REGION Network 145: PFE Maintenance Warnings_[Em5 → Em9]
   RUNG wire#powerrail
      Contact( "Unit1.Alarms".NoDataTransfer[12] )
      { S7_Templates := "time_type := Time" } "Unit1.Alarms".tonMaintenanceWarning[52].TON(pt := #DelayTime, et =>)
      Coil( "Unit1.Alarms".maintenanceWarnings[52] )
   END_RUNG
   // the same network as SCL:
   "Unit1.Alarms".tonMaintenanceWarning[52].TON(IN := "Unit1.Alarms".NoDataTransfer[12], PT := #DelayTime);
   "Unit1.Alarms".maintenanceWarnings[52] := "Unit1.Alarms".tonMaintenanceWarning[52].Q;
END_REGION

REGION Network 146: PFE Maintenance Warnings_[Em9 → Em5]
   RUNG wire#powerrail
      Contact( "Unit1.Alarms".NoDataTransfer[13] )
      { S7_Templates := "time_type := Time" } "Unit1.Alarms".tonMaintenanceWarning[53].TON(pt := #DelayTime, et =>)
      Coil( "Unit1.Alarms".maintenanceWarnings[53] )
   END_RUNG
   // the same network as SCL:
   "Unit1.Alarms".tonMaintenanceWarning[53].TON(IN := "Unit1.Alarms".NoDataTransfer[13], PT := #DelayTime);
   "Unit1.Alarms".maintenanceWarnings[53] := "Unit1.Alarms".tonMaintenanceWarning[53].Q;
END_REGION

REGION Network 147: PFE Maintenance Warnings_[Em5 → Em10]
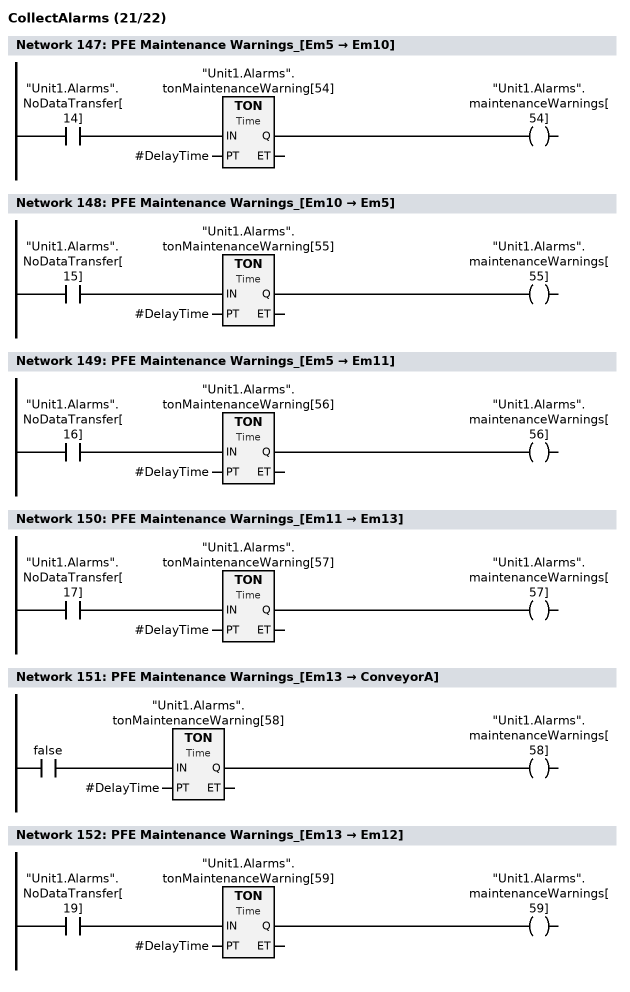
   RUNG wire#powerrail
      Contact( "Unit1.Alarms".NoDataTransfer[14] )
      { S7_Templates := "time_type := Time" } "Unit1.Alarms".tonMaintenanceWarning[54].TON(pt := #DelayTime, et =>)
      Coil( "Unit1.Alarms".maintenanceWarnings[54] )
   END_RUNG
   // the same network as SCL:
   "Unit1.Alarms".tonMaintenanceWarning[54].TON(IN := "Unit1.Alarms".NoDataTransfer[14], PT := #DelayTime);
   "Unit1.Alarms".maintenanceWarnings[54] := "Unit1.Alarms".tonMaintenanceWarning[54].Q;
END_REGION

REGION Network 148: PFE Maintenance Warnings_[Em10 → Em5]
   RUNG wire#powerrail
      Contact( "Unit1.Alarms".NoDataTransfer[15] )
      { S7_Templates := "time_type := Time" } "Unit1.Alarms".tonMaintenanceWarning[55].TON(pt := #DelayTime, et =>)
      Coil( "Unit1.Alarms".maintenanceWarnings[55] )
   END_RUNG
   // the same network as SCL:
   "Unit1.Alarms".tonMaintenanceWarning[55].TON(IN := "Unit1.Alarms".NoDataTransfer[15], PT := #DelayTime);
   "Unit1.Alarms".maintenanceWarnings[55] := "Unit1.Alarms".tonMaintenanceWarning[55].Q;
END_REGION

REGION Network 149: PFE Maintenance Warnings_[Em5 → Em11]
   RUNG wire#powerrail
      Contact( "Unit1.Alarms".NoDataTransfer[16] )
      { S7_Templates := "time_type := Time" } "Unit1.Alarms".tonMaintenanceWarning[56].TON(pt := #DelayTime, et =>)
      Coil( "Unit1.Alarms".maintenanceWarnings[56] )
   END_RUNG
   // the same network as SCL:
   "Unit1.Alarms".tonMaintenanceWarning[56].TON(IN := "Unit1.Alarms".NoDataTransfer[16], PT := #DelayTime);
   "Unit1.Alarms".maintenanceWarnings[56] := "Unit1.Alarms".tonMaintenanceWarning[56].Q;
END_REGION

REGION Network 150: PFE Maintenance Warnings_[Em11 → Em13]
   RUNG wire#powerrail
      Contact( "Unit1.Alarms".NoDataTransfer[17] )
      { S7_Templates := "time_type := Time" } "Unit1.Alarms".tonMaintenanceWarning[57].TON(pt := #DelayTime, et =>)
      Coil( "Unit1.Alarms".maintenanceWarnings[57] )
   END_RUNG
   // the same network as SCL:
   "Unit1.Alarms".tonMaintenanceWarning[57].TON(IN := "Unit1.Alarms".NoDataTransfer[17], PT := #DelayTime);
   "Unit1.Alarms".maintenanceWarnings[57] := "Unit1.Alarms".tonMaintenanceWarning[57].Q;
END_REGION

REGION Network 151: PFE Maintenance Warnings_[Em13 → ConveyorA]
   RUNG wire#powerrail
      Contact( false )
      { S7_Templates := "time_type := Time" } "Unit1.Alarms".tonMaintenanceWarning[58].TON(pt := #DelayTime, et =>)
      Coil( "Unit1.Alarms".maintenanceWarnings[58] )
   END_RUNG
   // the same network as SCL:
   "Unit1.Alarms".tonMaintenanceWarning[58].TON(IN := false, PT := #DelayTime);
   "Unit1.Alarms".maintenanceWarnings[58] := "Unit1.Alarms".tonMaintenanceWarning[58].Q;
END_REGION

REGION Network 152: PFE Maintenance Warnings_[Em13 → Em12]
   RUNG wire#powerrail
      Contact( "Unit1.Alarms".NoDataTransfer[19] )
      { S7_Templates := "time_type := Time" } "Unit1.Alarms".tonMaintenanceWarning[59].TON(pt := #DelayTime, et =>)
      Coil( "Unit1.Alarms".maintenanceWarnings[59] )
   END_RUNG
   // the same network as SCL:
   "Unit1.Alarms".tonMaintenanceWarning[59].TON(IN := "Unit1.Alarms".NoDataTransfer[19], PT := #DelayTime);
   "Unit1.Alarms".maintenanceWarnings[59] := "Unit1.Alarms".tonMaintenanceWarning[59].Q;
END_REGION

REGION Network 153: *************** Status ***************************
END_REGION

REGION Network 154: PFE Maintenance Status
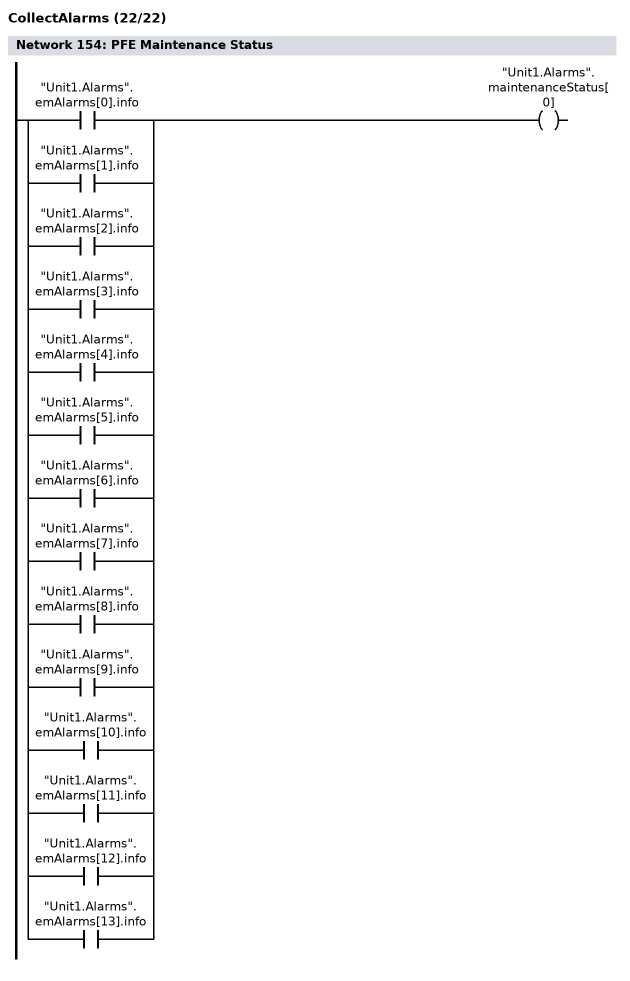
   RUNG wire#powerrail
      Contact( "Unit1.Alarms".emAlarms[0].info )
      wire#w1
      Coil( "Unit1.Alarms".maintenanceStatus[0] )
   END_RUNG
   RUNG wire#powerrail
      Contact( "Unit1.Alarms".emAlarms[1].info )
   END_RUNG wire#w1
   RUNG wire#powerrail
      Contact( "Unit1.Alarms".emAlarms[2].info )
   END_RUNG wire#w1
   RUNG wire#powerrail
      Contact( "Unit1.Alarms".emAlarms[3].info )
   END_RUNG wire#w1
   RUNG wire#powerrail
      Contact( "Unit1.Alarms".emAlarms[4].info )
   END_RUNG wire#w1
   RUNG wire#powerrail
      Contact( "Unit1.Alarms".emAlarms[5].info )
   END_RUNG wire#w1
   RUNG wire#powerrail
      Contact( "Unit1.Alarms".emAlarms[6].info )
   END_RUNG wire#w1
   RUNG wire#powerrail
      Contact( "Unit1.Alarms".emAlarms[7].info )
   END_RUNG wire#w1
   RUNG wire#powerrail
      Contact( "Unit1.Alarms".emAlarms[8].info )
   END_RUNG wire#w1
   RUNG wire#powerrail
      Contact( "Unit1.Alarms".emAlarms[9].info )
   END_RUNG wire#w1
   RUNG wire#powerrail
      Contact( "Unit1.Alarms".emAlarms[10].info )
   END_RUNG wire#w1
   RUNG wire#powerrail
      Contact( "Unit1.Alarms".emAlarms[11].info )
   END_RUNG wire#w1
   RUNG wire#powerrail
      Contact( "Unit1.Alarms".emAlarms[12].info )
   END_RUNG wire#w1
   RUNG wire#powerrail
      Contact( "Unit1.Alarms".emAlarms[13].info )
   END_RUNG wire#w1
   // the same network as SCL:
   "Unit1.Alarms".maintenanceStatus[0] := "Unit1.Alarms".emAlarms[0].info OR "Unit1.Alarms".emAlarms[1].info OR "Unit1.Alarms".emAlarms[2].info OR "Unit1.Alarms".emAlarms[3].info OR "Unit1.Alarms".emAlarms[4].info OR "Unit1.Alarms".emAlarms[5].info OR "Unit1.Alarms".emAlarms[6].info OR "Unit1.Alarms".emAlarms[7].info OR "Unit1.Alarms".emAlarms[8].info OR "Unit1.Alarms".emAlarms[9].info OR "Unit1.Alarms".emAlarms[10].info OR "Unit1.Alarms".emAlarms[11].info OR "Unit1.Alarms".emAlarms[12].info OR "Unit1.Alarms".emAlarms[13].info;
END_REGION
END_FUNCTION
